// TwinCAT 3 PLC project SIM
// ProgramVersion: 3.1.4024.0
// libraries:
//   Tc2_Standard, * (Beckhoff Automation GmbH)
//   Tc2_System, * (Beckhoff Automation GmbH)
//   Tc3_Module, * (Beckhoff Automation GmbH)
// project tree:
//   / PlcTask.TcTTO
//   POUs/Devices/ FB_SimActuator.TcPOU, FB_SimAxis.TcPOU
//   POUs/ FB_SimCell.TcPOU, MAIN.TcPOU
//   POUs/Stations/ FB_SimBarcodeScanner.TcPOU, FB_SimCheckWeigher.TcPOU, FB_SimFiller.TcPOU, FB_SimCapper.TcPOU
// (motion and I/O tree: see PLC project plc)
// real-time tasks:
//   TASK PlcTask: cycle T#10ms, priority 20, ADS port 350
// variable links:
//   PLC/PLC Instance <-> SIM/SIM Instance
//     PlcTask Inputs/MAIN.fbCell.bPartPresentAtInfeed <-> PlcTask Outputs/MAIN.fbSimCell.bPartPresentAtInfeed
//     PlcTask Inputs/MAIN.fbCell.bPartPresentAtOutfeed <-> PlcTask Outputs/MAIN.fbSimCell.bPartPresentAtOutfeed
//     PlcTask Inputs/MAIN.fbCell.fbBarcoder.bPartPresent <-> PlcTask Outputs/MAIN.fbSimCell.fbSimScanner.bPartPresent
//     PlcTask Inputs/MAIN.fbCell.fbBarcoder.sBarcode <-> PlcTask Outputs/MAIN.fbSimCell.fbSimScanner.sBarcode
//     PlcTask Inputs/MAIN.fbCell.fbCapper.bCapDone <-> PlcTask Outputs/MAIN.fbSimCell.fbSimCapper.bCapDone
//     PlcTask Inputs/MAIN.fbCell.fbCapper.bCapFail <-> PlcTask Outputs/MAIN.fbSimCell.fbSimCapper.bCapFail
//     PlcTask Inputs/MAIN.fbCell.fbCapper.bPartPresent <-> PlcTask Outputs/MAIN.fbSimCell.fbSimCapper.bPartPresent
//     PlcTask Inputs/MAIN.fbCell.fbCheckWeigher.bPartPresent <-> PlcTask Outputs/MAIN.fbSimCell.fbSimWeigher.bPartPresent
//     PlcTask Inputs/MAIN.fbCell.fbCheckWeigher.fScaleReading <-> PlcTask Outputs/MAIN.fbSimCell.fbSimWeigher.fScaleReading
//     PlcTask Inputs/MAIN.fbCell.fbFiller.bPartPresent <-> PlcTask Outputs/MAIN.fbSimCell.fbSimFiller.bPartPresent
//     PlcTask Inputs/MAIN.fbCell.fbFiller.fVolumeFilled <-> PlcTask Outputs/MAIN.fbSimCell.fbSimFiller.fVolumeFilled
//     PlcTask Inputs/MAIN.fbCell.fbIndexConveyor.bBusy <-> PlcTask Outputs/MAIN.fbSimCell.fbIndexConveyor.bBusy
//     PlcTask Inputs/MAIN.fbCell.fbIndexConveyor.bError <-> PlcTask Outputs/MAIN.fbSimCell.fbIndexConveyor.bError
//     PlcTask Inputs/MAIN.fbCell.fbIndexConveyor.bReady <-> PlcTask Outputs/MAIN.fbSimCell.fbIndexConveyor.bReady
//     PlcTask Inputs/MAIN.fbCell.fbIndexConveyor.bRunning <-> PlcTask Outputs/MAIN.fbSimCell.fbIndexConveyor.bRunning
//     PlcTask Inputs/MAIN.fbCell.fbIndexConveyor.fActPosition <-> PlcTask Outputs/MAIN.fbSimCell.fbIndexConveyor.fActPosition
//     PlcTask Inputs/MAIN.fbCell.fbIndexConveyor.fActVelocity <-> PlcTask Outputs/MAIN.fbSimCell.fbIndexConveyor.fActVelocity
//     PlcTask Inputs/MAIN.fbCell.fbInfeedActuator.bExtended <-> PlcTask Outputs/MAIN.fbSimCell.fbInfeedActuator.bExtended
//     PlcTask Inputs/MAIN.fbCell.fbInfeedActuator.bRetracted <-> PlcTask Outputs/MAIN.fbSimCell.fbInfeedActuator.bRetracted
//     PlcTask Inputs/MAIN.fbCell.fbInfeedConveyor.bBusy <-> PlcTask Outputs/MAIN.fbSimCell.fbInfeedConveyor.bBusy
//     PlcTask Inputs/MAIN.fbCell.fbInfeedConveyor.bError <-> PlcTask Outputs/MAIN.fbSimCell.fbInfeedConveyor.bError
//     PlcTask Inputs/MAIN.fbCell.fbInfeedConveyor.bReady <-> PlcTask Outputs/MAIN.fbSimCell.fbInfeedConveyor.bReady
//     PlcTask Inputs/MAIN.fbCell.fbInfeedConveyor.bRunning <-> PlcTask Outputs/MAIN.fbSimCell.fbInfeedConveyor.bRunning
//     PlcTask Inputs/MAIN.fbCell.fbInfeedConveyor.fActPosition <-> PlcTask Outputs/MAIN.fbSimCell.fbInfeedConveyor.fActPosition
//     PlcTask Inputs/MAIN.fbCell.fbInfeedConveyor.fActVelocity <-> PlcTask Outputs/MAIN.fbSimCell.fbInfeedConveyor.fActVelocity
//     PlcTask Inputs/MAIN.fbCell.fbOutfeedActuator.bExtended <-> PlcTask Outputs/MAIN.fbSimCell.fbOutfeedActuator.bExtended
//     PlcTask Inputs/MAIN.fbCell.fbOutfeedActuator.bRetracted <-> PlcTask Outputs/MAIN.fbSimCell.fbOutfeedActuator.bRetracted
//     PlcTask Inputs/MAIN.fbCell.fbOutfeedConveyor.bBusy <-> PlcTask Outputs/MAIN.fbSimCell.fbOutfeedConveyor.bBusy
//     PlcTask Inputs/MAIN.fbCell.fbOutfeedConveyor.bError <-> PlcTask Outputs/MAIN.fbSimCell.fbOutfeedConveyor.bError
//     PlcTask Inputs/MAIN.fbCell.fbOutfeedConveyor.bReady <-> PlcTask Outputs/MAIN.fbSimCell.fbOutfeedConveyor.bReady
//     PlcTask Inputs/MAIN.fbCell.fbOutfeedConveyor.bRunning <-> PlcTask Outputs/MAIN.fbSimCell.fbOutfeedConveyor.bRunning
//     PlcTask Inputs/MAIN.fbCell.fbOutfeedConveyor.fActPosition <-> PlcTask Outputs/MAIN.fbSimCell.fbOutfeedConveyor.fActPosition
//     PlcTask Inputs/MAIN.fbCell.fbOutfeedConveyor.fActVelocity <-> PlcTask Outputs/MAIN.fbSimCell.fbOutfeedConveyor.fActVelocity
//     PlcTask Outputs/MAIN.fbCell.fFillRate <-> PlcTask Inputs/MAIN.fbSimCell.fFillRate
//     PlcTask Outputs/MAIN.fbCell.fbBarcoder.bTriggerRead <-> PlcTask Inputs/MAIN.fbSimCell.fbSimScanner.bTriggerRead
//     PlcTask Outputs/MAIN.fbCell.fbCapper.bCapTrigger <-> PlcTask Inputs/MAIN.fbSimCell.fbSimCapper.bCapTrigger
//     PlcTask Outputs/MAIN.fbCell.fbCapper.bClamp <-> PlcTask Inputs/MAIN.fbSimCell.fbSimCapper.bClamp
//     PlcTask Outputs/MAIN.fbCell.fbCheckWeigher.bLift <-> PlcTask Inputs/MAIN.fbSimCell.fbSimWeigher.bLift
//     PlcTask Outputs/MAIN.fbCell.fbFiller.bFillValve <-> PlcTask Inputs/MAIN.fbSimCell.fbSimFiller.bFillValve
//     PlcTask Outputs/MAIN.fbCell.fbIndexConveyor.bJogFwdCmd <-> PlcTask Inputs/MAIN.fbSimCell.fbIndexConveyor.bJogFwdCmd
//     PlcTask Outputs/MAIN.fbCell.fbIndexConveyor.bMoveAbsCmd <-> PlcTask Inputs/MAIN.fbSimCell.fbIndexConveyor.bMoveAbsCmd
//     PlcTask Outputs/MAIN.fbCell.fbIndexConveyor.fPositionCmd <-> PlcTask Inputs/MAIN.fbSimCell.fbIndexConveyor.fPositionCmd
//     PlcTask Outputs/MAIN.fbCell.fbIndexConveyor.fVelocityCmd <-> PlcTask Inputs/MAIN.fbSimCell.fbIndexConveyor.fVelocityCmd
//     PlcTask Outputs/MAIN.fbCell.fbInfeedActuator.bExtendCmd <-> PlcTask Inputs/MAIN.fbSimCell.fbInfeedActuator.bExtendCmd
//     PlcTask Outputs/MAIN.fbCell.fbInfeedActuator.bRetractCmd <-> PlcTask Inputs/MAIN.fbSimCell.fbInfeedActuator.bRetractCmd
//     PlcTask Outputs/MAIN.fbCell.fbInfeedConveyor.bJogFwdCmd <-> PlcTask Inputs/MAIN.fbSimCell.fbInfeedConveyor.bJogFwdCmd
//     PlcTask Outputs/MAIN.fbCell.fbInfeedConveyor.bMoveAbsCmd <-> PlcTask Inputs/MAIN.fbSimCell.fbInfeedConveyor.bMoveAbsCmd
//     PlcTask Outputs/MAIN.fbCell.fbInfeedConveyor.fPositionCmd <-> PlcTask Inputs/MAIN.fbSimCell.fbInfeedConveyor.fPositionCmd
//     PlcTask Outputs/MAIN.fbCell.fbInfeedConveyor.fVelocityCmd <-> PlcTask Inputs/MAIN.fbSimCell.fbInfeedConveyor.fVelocityCmd
//     PlcTask Outputs/MAIN.fbCell.fbOutfeedActuator.bExtendCmd <-> PlcTask Inputs/MAIN.fbSimCell.fbOutfeedActuator.bExtendCmd
//     PlcTask Outputs/MAIN.fbCell.fbOutfeedActuator.bRetractCmd <-> PlcTask Inputs/MAIN.fbSimCell.fbOutfeedActuator.bRetractCmd
//     PlcTask Outputs/MAIN.fbCell.fbOutfeedConveyor.bJogFwdCmd <-> PlcTask Inputs/MAIN.fbSimCell.fbOutfeedConveyor.bJogFwdCmd
//     PlcTask Outputs/MAIN.fbCell.fbOutfeedConveyor.bMoveAbsCmd <-> PlcTask Inputs/MAIN.fbSimCell.fbOutfeedConveyor.bMoveAbsCmd
//     PlcTask Outputs/MAIN.fbCell.fbOutfeedConveyor.fPositionCmd <-> PlcTask Inputs/MAIN.fbSimCell.fbOutfeedConveyor.fPositionCmd
//     PlcTask Outputs/MAIN.fbCell.fbOutfeedConveyor.fVelocityCmd <-> PlcTask Inputs/MAIN.fbSimCell.fbOutfeedConveyor.fVelocityCmd

CONFIGURATION SIM
    RESOURCE PLC ON TwinCAT3
        TASK PlcTask(INTERVAL := T#10ms, PRIORITY := 20);
        PROGRAM MAIN WITH PlcTask : MAIN;
    END_RESOURCE
END_CONFIGURATION

// ---- POUs/MAIN.TcPOU
PROGRAM MAIN
VAR
	fbSimCell		: FB_SimCell;
	Seed			: INT;
END_VAR

Seed := Seed + 1;
fbSimCell();

END_PROGRAM

// ---- POUs/FB_SimCell.TcPOU
FUNCTION_BLOCK FB_SimCell
VAR_INPUT
END_VAR
VAR_OUTPUT
END_VAR
VAR
	bPartPresentAtInfeed		AT %Q* : BOOL;
	bPartPresentAtOutfeed		AT %Q* : BOOL;
	fFillRate					AT %I* : LREAL;
	
	fbInfeedActuator			: FB_SimActuator;
	fbOutfeedActuator			: FB_SimActuator;
	fbInfeedConveyor			: FB_SimAxis;
	fbOutfeedConveyor			: FB_SimAxis;
	fbIndexConveyor				: FB_SimAxis;
	
	fbSimScanner				: FB_SimBarcodeScanner;
	fbSimFiller					: FB_SimFiller;
	fbSimCapper					: FB_SimCapper;
	fbSimWeigher				: FB_SimCheckWeigher;
	
	fbTmr						: ARRAY[0..9] OF TON;
	rand						: ARRAY[0..9] OF DRAND;
	i,j,k						: INT;
	bStationLoaded				: ARRAY[0..3] OF BOOL;
	fFillAmount					: ARRAY[0..2] OF LREAL;
	
	iIndexState					: DINT;
	iInfeedState				: DINT;
	iOutfeedState				: DINT;
END_VAR

FOR i := 0 TO 9 DO
	rand[i](Seed:=MAIN.Seed+i);
END_FOR

fbInfeedActuator();
fbInfeedConveyor();
fbIndexConveyor();
fbOutfeedActuator();
fbOutfeedConveyor();

fbSimScanner();
fbSimFiller(fFillRate:=fFillRate, fFillAmount=>fFillAmount[0]);
fbSimCapper();
fbSimWeigher(fFillAmount:=fFillAmount[2]);

// Infeed
CASE iInfeedState OF
	0:
		fbTmr[0].PT := TO_TIME(1000 + rand[0].Num * 1000);
		iInfeedState := 1;
		
	1:
		fbTmr[0](IN:=(fbInfeedConveyor.State <> 0 AND NOT bPartPresentAtInfeed));
		IF fbTmr[0].Q THEN
			fbTmr[0](IN:=FALSE);
			bPartPresentAtInfeed := TRUE;
			iInfeedState := 2;
		END_IF
		
	2:
		IF fbInfeedActuator.bExtended THEN
			bPartPresentAtInfeed := FALSE;
			fbSimScanner.PartPresent := TRUE;
			bStationLoaded[0] := TRUE;
			iInfeedState := 3;
		END_IF
	
	3:
		iInfeedState := 0;
		
END_CASE


CASE iIndexState OF
	0:
		// conveyor indexing
		IF fbIndexConveyor.bMoveAbsCmd AND 
			(fbIndexConveyor.fActPosition <> fbIndexConveyor.fPositionCmd) THEN
			iIndexState := 1;
		END_IF
		
	1:
		fbSimScanner.PartPresent := FALSE;
		fbSimFiller.PartPresent := FALSE;
		fbSimCapper.PartPresent := FALSE;
		fbSimWeigher.PartPresent := FALSE;
		
		// index complete
		IF fbIndexConveyor.fActPosition = fbIndexConveyor.fPositionCmd THEN
			iIndexState := 2;
		END_IF
		
	2:
		// shift parts
		fbSimScanner.PartPresent := FALSE;
		fbSimFiller.PartPresent := bStationLoaded[0];
		fbSimCapper.PartPresent := bStationLoaded[1];
		fbSimWeigher.PartPresent := bStationLoaded[2];
		bPartPresentAtOutfeed := bStationLoaded[3];
		
		fFillAmount[2] := fFillAmount[1];
		fFillAmount[1] := fFillAmount[0];
		
		bStationLoaded[3] := bStationLoaded[2];
		bStationLoaded[2] := bStationLoaded[1];
		bStationLoaded[1] := bStationLoaded[0];
		bStationLoaded[0] := FALSE;
		
		iIndexState := 0;
		
END_CASE

// Outfeed
CASE iOutfeedState OF
	0:
		fbTmr[1](IN:=FALSE);
		IF bPartPresentAtOutfeed THEN
			iOutFeedState := 1;
		END_IF
		
	1:
		fbTmr[1](IN:=TRUE, PT:=T#3S);
		IF fbTmr[1].Q THEN
			bPartPresentAtOutfeed := FALSE;
			iOutfeedState := 0;
		END_IF
		
		IF fbOutfeedActuator.bExtended THEN
			bPartPresentAtOutfeed := FALSE;
			iOutfeedState := 0;
		END_IF
		
END_CASE

END_FUNCTION_BLOCK

// ---- POUs/Devices/FB_SimActuator.TcPOU
FUNCTION_BLOCK FB_SimActuator
VAR_INPUT
END_VAR
VAR_OUTPUT
END_VAR
VAR
	bExtended			AT %Q* : BOOL;
	bRetracted			AT %Q* : BOOL := TRUE;
	bExtendCmd			AT %I* : BOOL;
	bRetractCmd			AT %I* : BOOL;
	
	State				: DINT;
	tmrExtend			: TON;
	tmrRetract			: TON;
	iExtendMs			: DINT;
	iRetractMs			: DINT;
	rand				: DRAND;
END_VAR

rand(Seed:=TO_INT(iExtendMs + iRetractMs));
CASE State OF
	0:
		IF bExtendCmd THEN
			iExtendMs := TO_DINT(1500 + (rand.Num * 500));
			State := 1;
		END_IF
		
		IF bRetractCmd THEN
			iRetractMs := TO_DINT(1500 + (rand.Num * 500));
			State := 2;
		END_IF
		
	1:
		tmrExtend(IN:=TRUE, PT:=TO_TIME(iExtendMs));
		IF TO_DINT(tmrExtend.PT) > rand.Num * 100 THEN
			bRetracted := FALSE;
		END_IF
		IF tmrExtend.Q THEN
			bExtended := TRUE;
			tmrExtend(IN:=FALSE);
			State := 0;
		END_IF
		
	2:
		tmrRetract(IN:=TRUE, PT:=TO_TIME(iRetractMs));
		IF TO_DINT(tmrRetract.PT) > rand.Num * 100 THEN
			bExtended := FALSE;
		END_IF
		IF tmrRetract.Q THEN
			bRetracted := TRUE;
			tmrRetract(IN:=FALSE);
			State := 0;
		END_IF
		
END_CASE

END_FUNCTION_BLOCK

// ---- POUs/Devices/FB_SimAxis.TcPOU
FUNCTION_BLOCK FB_SimAxis
VAR_INPUT
END_VAR
VAR_OUTPUT
END_VAR
VAR
	fActPosition			AT %Q* : LREAL;
	fActVelocity			AT %Q* : LREAL;
	bReady					AT %Q* : BOOL := TRUE;
	bBusy					AT %Q* : BOOL;
	bError					AT %Q* : BOOL;
	bRunning				AT %Q* : BOOL;
	
	fPositionCmd			AT %I* : LREAL;
	fVelocityCmd			AT %I* : LREAL;
	bJogFwdCmd				AT %I* : BOOL;
	bMoveAbsCmd				AT %I* : BOOL;
	
	State					: DINT;
	fVelocity				: LREAL;
END_VAR

fVelocity := fVelocityCmd / 100.177;

CASE State OF
	0:
		bReady := TRUE;
		bBusy := FALSE;
		bRunning := FALSE;
		bError := FALSE;
		
		IF bJogFwdCmd THEN
			State := 10;
		END_IF
		
		IF bMoveAbsCmd AND (fActPosition <> fPositionCmd) THEN
			State := 20;
		END_IF
		
	10:
		bBusy := TRUE;
		bRunning := TRUE;
		bReady := FALSE;
		fActVelocity := fVelocityCmd;
		fActPosition := fActPosition + fVelocity;
		IF NOT bJogFwdCmd THEN
			State := 0;
		END_IF
		
	20:
		bBusy := TRUE;
		bRunning := TRUE;
		bReady := FALSE;
		IF fPositionCmd > fActPosition THEN
			State := 21;
		ELSE
			State := 22;
		END_IF
		
	21:
		IF (fPositionCmd > fActPosition) THEN
			fActPosition := fActPosition + fVelocity;
		ELSE
			fActPosition := fPositionCmd;
			State := 0;
		END_IF
		IF NOT bMoveAbsCmd THEN
			State := 0;
		END_IF
	
	22:
		fActVelocity := -(fVelocityCmd);
		IF (fPositionCmd < fActPosition) THEN
			fActPosition := fActPosition - fVelocity;
		ELSE
			fActPosition := fPositionCmd;
			State := 0;
		END_IF
		IF NOT bMoveAbsCmd THEN
			State := 0;
		END_IF
	
END_CASE

END_FUNCTION_BLOCK

// ---- POUs/Stations/FB_SimBarcodeScanner.TcPOU
FUNCTION_BLOCK FB_SimBarcodeScanner
VAR_INPUT
END_VAR
VAR_OUTPUT
END_VAR
VAR
	bTriggerRead				AT %I* : BOOL;
	sBarcode					AT %Q* : STRING(255);
	
	rand						: DRAND;
	fRand						: LREAL;
	tmrWork						: TON;
	iWorkMs						: DINT;
	iState						: DINT;
END_VAR
VAR CONSTANT
	CHANCE_NOREAD				: LREAL := 0.05;
	NO_READ						: STRING(255) := 'NO_READ';
END_VAR

rand(Seed:=107);

CASE iState OF
	0:
		IF bTriggerRead THEN
			fRand := rand.Num;
			iWorkMs := 250 + TO_DINT(fRand * 1000);
			iState := 10;
		ELSE
			sBarcode := '';
		END_IF
		
	10:
		tmrWork(IN:=TRUE, PT:=TO_TIME(iWorkMs));
		IF tmrWork.Q THEN
			tmrWork(IN:=FALSE);
			IF rand.Num > CHANCE_NOREAD THEN
				sBarcode := CONCAT('BRCD_', TO_STRING(TO_DINT(fRand * 100000)));
			ELSE
				sBarcode := NO_READ;
			END_IF
			iState := 20;
		END_IF
		
	20:
		iState := 0;
		
END_CASE

END_FUNCTION_BLOCK

// ---- POUs/Stations/FB_SimFiller.TcPOU
FUNCTION_BLOCK FB_SimFiller
VAR_INPUT
END_VAR
VAR_OUTPUT
END_VAR
VAR
	fVolumeFilled				AT %Q* : LREAL;
	bFillValve					AT %I* : BOOL;
	
	rand						: DRAND;
	iState						: DINT;
END_VAR
VAR CONSTANT
	FLOW_RATE					: LREAL := 1.0;
END_VAR

rand(Seed:=113);

CASE iState OF
	0:
		IF bFillValve THEN
			iState := 10;
		ELSE
			fVolumeFilled := 0.0;
		END_IF
		
	10:
		IF bFillValve THEN
			fVolumeFilled := fVolumeFilled + (FLOW_RATE + rand.Num);
		ELSE
			iState := 20;
		END_IF
		
	20:
		iState := 0;
		
END_CASE

END_FUNCTION_BLOCK

// ---- POUs/Stations/FB_SimCapper.TcPOU
FUNCTION_BLOCK FB_SimCapper
VAR_INPUT
END_VAR
VAR_OUTPUT
END_VAR
VAR
	bClamp						AT %I* : BOOL;
	bCapTrigger					AT %I* : BOOL;
	bCapDone					AT %Q* : BOOL;
	bCapFail					AT %Q* : BOOL;
	
	rand						: DRAND;
	iCapMs						: DINT;
	tmrCap						: TON;
	iState						: DINT;
END_VAR
VAR CONSTANT
	CHANCE_FAIL					: LREAL := 0.01;
END_VAR

rand(Seed:=117);

CASE iState OF
	0:
		IF bCapTrigger THEN
			iState := 10;
			iCapMs := 1000 + TO_DINT(rand.Num * 100);
		ELSE
			bCapDone := FALSE;
			bCapFail := FALSE;
		END_IF
		
	10:
		tmrCap(IN:=TRUE, PT:=TO_TIME(iCapMs));
		IF tmrCap.Q THEN
			tmrCap(IN:=FALSE);
			IF rand.Num < CHANCE_FAIL THEN
				bCapFail := TRUE;
			END_IF
			bCapDone := TRUE;
			iState := 20;
		END_IF
		
	20:
		iState := 0;
		
END_CASE

END_FUNCTION_BLOCK

// ---- POUs/Stations/FB_SimCheckWeigher.TcPOU
FUNCTION_BLOCK FB_SimCheckWeigher
VAR_INPUT
END_VAR
VAR_OUTPUT
END_VAR
VAR
	bLift						AT %I* : BOOL;
	fScaleReading				AT %Q* : LREAL;
	
	rand						: DRAND;
	fWeightSetpoint				: LREAL;
	tmrWork						: TON;
	iWorkMs						: DINT;
	iState						: DINT;
END_VAR

rand(Seed:=123);

CASE iState OF
	0:
		IF bLift THEN
			iState := 10;
		ELSE
			fScaleReading := 0.0 + (rand.Num / 1000);
		END_IF

	10:
		IF fScaleReading < fWeightSetpoint THEN
			fScaleReading := fScaleReading + (fWeightSetpoint / 5) + (rand.Num * 10);
		ELSE
			iState := 20;
		END_IF
		
	20:
		IF NOT bLift THEN
			IF fScaleReading < fWeightSetpoint THEN
				fScaleReading := fScaleReading + (rand.Num / 1000);
			ELSE
				fScaleReading := fScaleReading - (rand.Num / 1000);
			END_IF
		ELSE
			iState := 0;
		END_IF
		
END_CASE

END_FUNCTION_BLOCK
